// TIA Portal V16 export
// export: Created 2024-09-05T15:58:42.4292171Z, ExportSetting WithDefaults, DisplayName Totally Integrated Automation Portal, DisplayVersion V16 Update 6, DisplayName TIA Portal Version Control Interface, DisplayVersion V16 Update 2, DisplayName TIA Portal Openness, DisplayVersion V16 Update 6, DisplayName STEP 7 Professional, DisplayVersion V16 Update 6, DisplayName STEP 7 Safety, DisplayVersion V16, DisplayName WinCC Advanced, DisplayVersion V16 Update 6
VAR_GLOBAL   // PLC tag table "autoeject"
   iAEtubePresentFront AT %I35.0 : Bool;
   iAEtubePresentRear AT %I35.1 : Bool;
   i4partPresent AT %I27.3 : Bool;   // ok position
END_VAR
